FUNCTION_BLOCK T_ModuleCollectionSetSubModuleInfoCountGreaterThanSubModulesReturnError EXTENDS T_UnitTestBase
VAR
  list : T_SubModuleCollection;
  newModule, newModule2, newModule3 : T_SubModuleMock; 
  result : BOOL;
  
  PMLSubModuleInfo  : ARRAY[1..2] OF ST_PMLSubUnitInfo;
END_VAR

// Arrange
result := TRUE;
list.AddModule(newModule);
list.AddModule(newModule2);
list.AddModule(newModule3);

//Act
result := list.SetPMLSubModuleInfoActive(PMLSubModuleInfo);

//Assert
assertion.AssertEquals_BOOL(FALSE, result, 'NOT list.SetPMLSubModuleInfoActive(PMLSubModuleInfo)');
TestFinished();

END_FUNCTION_BLOCK

(* stored: Version 1.1.0.1, ProductVersion 3.1.4024.12
   POU T_ModuleCollectionSetSubModuleInfoCountGreaterThanSubModulesReturnError: Id {51ab96ba-1931-4a81-b02d-30462115a89b}, SpecialFunc None *)
